RoboDK station: UR10e.rdk

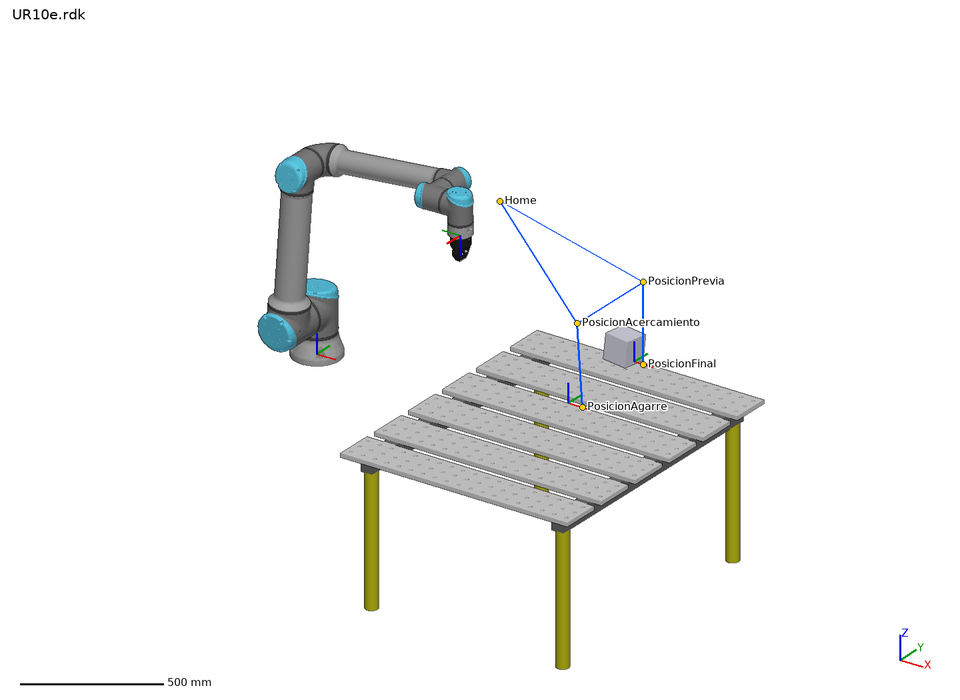
[picture v0: the station drawn from its stored meshes, robots at their saved joint values, targets as dots, program paths as lines]
Station Clase1IndustrialRobotics (saved by RoboDK 5.5.2). Poses are relative to the parent item; angles as X-Y-Z fixed-axis rotations.
  - frame UR10e Base at (0, 0, 0) mm
    - robot UR10e: 6 axes, payload 10 kg, reach 1300 mm, repeatability 0.05 mm, weight 28.9 kg
        modified DH rows (alpha deg, a mm, theta deg, d mm): 0, 0, 0, 180.7; 90, 0, 180, 0; 0, 612.6, 0, 0; 0, 571.335, 0, 174.15; -90, 0, 0, 119.85; 90, 0, 180, 116.55
        joint limits [-360, -360, -360, -360, -360, -360] to [360, 360, 360, 360, 360, 360]; home [0, -90, -90, 0, 90, 0]; saved at [-0.149, -94.095, -80.252, -94.407, 89.966, 1.561]
      - frame RobotiQ 2F85 Base at (0, 0, 0) mm
        - robot RobotiQ 2F85: 1 axes, payload 5 kg
            joint limits [0] to [85]; home [85]; saved at [85]
        - target Open (Cartesian target) at (938.55, 100, 246.18) mm, rotated rx -85.99 ry 0 rz -90 deg; joints [85] of RobotiQ 2F85
        - target Close (Cartesian target) at (0, 0, 103.92) mm; joints [68.98] of RobotiQ 2F85
      - tool 2F85, TCP at (0, 0, 211.5) mm
    - target PosicionAgarre (Cartesian target) at (1059.85, 100, 50) mm, rotated rx -85.99 ry 0 rz -90 deg; joints [21.396, -153.863, -98.022, 76.192, 68.659, -1.57] of UR10e
    - target Home (Cartesian target) at (899.38, -174.15, 913.15) mm, rotated rx -90 ry 0 rz -90 deg; joints [0, -90, -90, 0, 90, 0] of UR10e
    - target PosicionAcercamiento (Cartesian target) at (1037.47, 100, 369.22) mm, rotated rx -85.99 ry 0 rz -90 deg; joints [22.067, -125.528, -106.843, 56.698, 67.99, -1.624] of UR10e
    - target PosicionPrevia (Cartesian target) at (1037.47, 500, 369.22) mm, rotated rx -85.99 ry 0 rz -90 deg; joints [46.712, -135.658, -86.279, 47.776, 43.437, -4.247] of UR10e
    - target PosicionFinal (Cartesian target) at (1037.47, 500, 50) mm, rotated rx -85.99 ry 0 rz -90 deg; joints [46.712, -159.071, -80.316, 65.226, 43.437, -4.247] of UR10e
  - object Table at (1000, 0, 0) mm, rotated rx 0 ry 0 rz 90 deg, size 1193.8 x 965.2 x 609.6 mm, geometry from welding_table.sld
  - frame PosicionA at (1000, 100, 50) mm
  - frame PosicionB at (1000, 500, 50) mm
    - object box at (-40.58, -3.89, 50) mm, rotated rx -4.01 ry 3.72 rz -4.28 deg, size 100 x 100 x 100 mm, geometry from box.sld
  - program ProgramaPrincipal (14 instructions, listed below)
  - Python program CinematicaInversaConGripper (listed below)
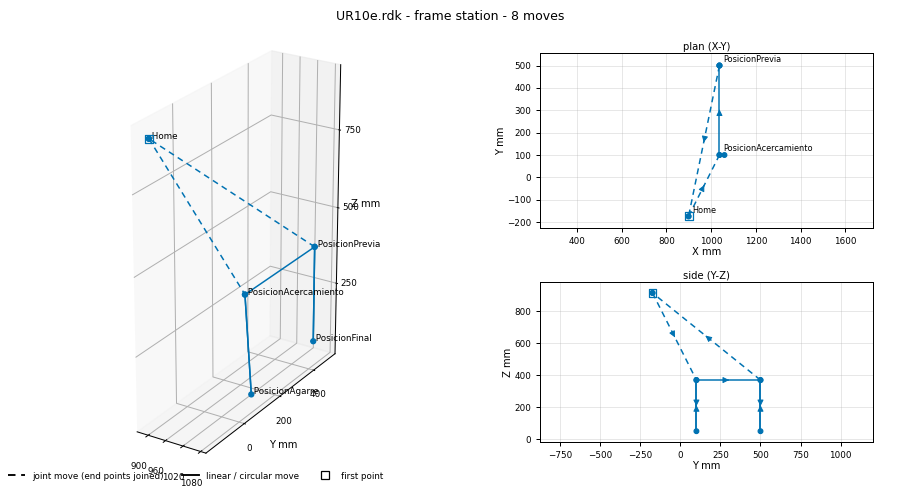
[picture p0: tool path of UR10e.rdk in frame station, 8 of 8 moves have a stored position in this frame; points joined in program order, loops and branches not executed]

--- program ProgramaPrincipal (robot UR10e) ---
  Est. Ref.: UR10e Base
  Est. herr: 2F85
  MoveJ (Home)
  MoveJ (PosicionAcercamiento)
  MoveL (PosicionAgarre)
  Adjuntar a 2F85
  MoveL (PosicionAcercamiento)
  Establecer velocidad (50.0 mm/s)
  MoveL (PosicionPrevia)
  MoveL (PosicionFinal)
  Separar de 2F85
  MoveL (PosicionPrevia)
  Establecer velocidad (500.0 mm/s)
  MoveJ (Home)

--- Python program CinematicaInversaConGripper ---
import math

import numpy as np
from robodk import *
from robolink import *  # RoboDK API
"""
import robotiq_gripper

#from numpy.linalg import inv
#import time

#Funciones para gripper (NO ALTERAR)
def log_info(gripper):
    print(f"Pos: {str(gripper.get_current_position()): >3} "
          f"Open: {gripper.is_open(): <2} "
          f"Closed: {gripper.is_closed(): <2} ")


def dt_gripper_position(current_position): #(NO ALTERAR)
    dt_pos = [0]
    dt_pos[0] = 85 - (current_position / gMax_Pos) * 85
    return dt_pos
"""
# Function to move real gripper and see it in RoboDK simulation (Open) (NO ALTERAR)
def open_gripper():
    if RDK.RunMode() > 1:
        RDK.setRunMode(1) #Set RunMode to see movement in robot and simulation
    time.sleep(0.5)
    gripper.move_and_wait_for_pos(int(gMin_Pos), 255, 255) #Move real gripper
    log_info(gripper) #Print info about gripper position
    dt_pos = dt_gripper_position(gripper.get_current_position()) # give actual position of gripper in milimeters
    dt_gripper.MoveJ(dt_pos) #move simulated gripper
    time.sleep(0.5)
    RDK.setRunMode(6) #Set Run mode to PC-Real Robot connection
    time.sleep(0.5)

# Function to move real gripper and see it in RoboDK simulation (Close) (NO ALTERAR)
def close_gripper():
    if RDK.RunMode() > 1:
        RDK.setRunMode(1)
    gripper.move_and_wait_for_pos(int(gMax_Pos), 255, 191)
    log_info(gripper)
    dt_pos = dt_gripper_position(gripper.get_current_position())
    dt_gripper.MoveJ(dt_pos)
    #input("Press 'Enter' to continue...")
    gripper.move_and_wait_for_pos(gMax_Pos, 255, 191)
    log_info(gripper)
    dt_pos = dt_gripper_position(gripper.get_current_position())
    dt_gripper.MoveJ(dt_pos)
    #input("Press 'Enter' to continue...")
    time.sleep(0.5)
    RDK.setRunMode(6)
    time.sleep(0.5)

#Suministar los datos de posicion y rotacion ROLL PITCH YAW
#TCP: Vector Tool Pose
#X : Posicion en X -- en milimetros [mm]
#Y : Posicion en Y -- en milimetros [mm]
#Z : Posicion en Z -- en milimetros [mm]
#RX : Rotacion en X - Yaw -- En grados [°]
#RY : Rotacion en Y - Pitch -- En grados [°]
#RZ : Rotacion en Z - Roll -- En grados [°]
#VTCP = [X,Y,Z,RX,RY,RZ]

VTCP=[1000,300,500,90,-90,90] #Ejemplo

#Conexion a RoboDK y robot
robot_ip = "192.168.1.10"  # Replace with your robot ip
rdk_ip = 'localhost'  # Or the explicit ip of the computer running RoboDK
### Connect to the RoboDK API ###
RDK = Robolink(robodk_ip=rdk_ip, port=20500)

rdk_robot = RDK.Item('UR10e')  # retrieve the robot by name
dt_gripper = RDK.Item('RobotiQ 2F85')  # the robotiq gripper inside RoboDK, It is not TCP attached to robot

"""
#Este codigo es ESENCIAL para asegurar la conexion al robot
status, status_msg = rdk_robot.ConnectedState()
while status != ROBOTCOM_READY:
    print(status_msg)
    rdk_robot.Disconnect()
    time.sleep(2)
    try:
        success = rdk_robot.Connect(robot_ip=robot_ip) ##IP UR10e PolyScope
        #success = Robot.Connect(robot_ip="192.168.1.10") ##IP UR10e real
        status, status_msg = rdk_robot.ConnectedState()
    except e:
        print(status_msg)
    if status == ROBOTCOM_READY:
        break

# Uses robotiq_gripper class to connect to gripper via sockets
print("Creating gripper...")
gripper = robotiq_gripper.RobotiqGripper()
print("Connecting to gripper...")
gripper.connect(robot_ip, 63352)  # The port on the URe family is 63352
print("Activating gripper...")
# When this executes the gripper will close and open again. Be careful.
# This function gets the max and min values of the gripper
gripper.activate()
# The gripper not always closes using the default max. It depends on the calibration
# So its is useful to know the current max of the system
gMax_Pos = gripper.get_max_position() #Fully Close
gMin_Pos = gripper.get_min_position() #Fully Open
"""
#Longitudes de links
d1= 180.7 #En milimetros
a2 = -612.7 #En mm
a3= -571.55 #En mm
d4= 174.15 #En mm
d5= 119.85 #En mm
d6= 116.55+211.5 #En mm. Se suma el valor del TCP de la herramienta

#Inserte algoritmo de cinematica inversa
def sen(grados):
    return math.sin(math.radians(grados))

def cos(grados):
    return math.cos(math.radians(grados))

def CInversa(VTCP):
    PX=VTCP[0]
    PY=VTCP[1]
    PZ=VTCP[2]
    Psi=VTCP[3]
    Theta=VTCP[4]
    phi=VTCP[5]
    T=np.array([[cos(phi)*cos(Theta),(sen(Psi)*cos(phi)*sen(Theta))-(cos(Psi)*sen(phi)),(sen(Psi)*sen(phi))+(cos(Psi)*cos(phi)*sen(Theta)),PX],
                [cos(Theta)*sen(phi), (cos(Psi)*cos(phi))+(sen(Psi)*sen(phi)*sen(Theta)),(cos(Psi)*sen(phi)*sen(Theta))-(sen(Psi)*cos(phi)),PY],
                [-sen(Theta),sen(Psi)*cos(Theta),cos(Psi)*cos(Theta),PZ],
                [0, 0, 0, 1]])
    for i in range(4):
        for j in range(4):
            T[i][j]=round(T[i][j],2)

    #Calculo del angulo theta1
    #Vector posicion de 0 a 5
    Z06=[T[0][2],T[1][2],T[2][2]]
    P06=[T[0][3],T[1][3],T[2][3]]
    P05=P06-np.dot(d6,Z06) #Se resta a la posicion en el SC6 la distancia al SC5 considerando la rotacion Z06
    phi1=math.degrees(math.atan2(P05[1],P05[0]))
    P05XY=math.sqrt(math.pow(P05[1],2)+math.pow(P05[0],2))
    phi2=math.degrees(math.acos(d4/P05XY))
    theta1=phi1+phi2+90
    theta1=round(theta1,2)
    #INICIO DE CODIGO DE CINEMATICA INVERSA (Del Angulo 2 al 6)
    theta5=math.degrees(math.acos((P06[0]*sen(theta1)-P06[1]*cos(theta1)-d4)/d6))
    CT6=math.degrees(-T[1][0]*sen(theta1)+(T[1][1]*cos(theta1))/sen(theta5))
    ST6=math.degrees(T[0][0]*sen(theta1)-(T[0][1]*cos(theta1))/sen(theta5))
    theta6=math.degrees(math.atan2(CT6,ST6))
    T1=np.array([[cos(theta1),0,sen(theta1),0],[sen(theta1),0,-cos(theta1),0],[0,1,0,d1],[0,0,0,1]])
    T5=np.array([[cos(theta5),0,-sen(theta5),0],[sen(theta5),0,cos(theta5),0],[0,-1,0,d5],[0,0,0,1]])
    T6=np.array([[cos(theta6),-sen(theta6),0,0],[sen(theta6),cos(theta6),0,0],[0,0,1,d6],[0,0,0,1]])
    P45=T5
    P56=T6
    P46=np.dot(P45,P56)
    P64=np.linalg.inv(P46)
    P10=np.linalg.inv(T1)
    P16=np.dot(P10,T)
    P14=np.dot(P16,P64)
    P14XY=math.sqrt((math.pow(P14[1][3],2))+math.pow(P14[0][3],2))
    theta3=math.degrees(math.acos(((P14XY**2)-(a2**2)-(a3**2))/(2*a2*a3)))
    theta2=(math.degrees(math.atan2(-P14[1][3],-P14[0][3])))-math.degrees(math.asin(-a3*sen(theta3)/P14XY))
    T2=np.array([[cos(theta2),-sen(theta2),0,a2*cos(theta2)],[sen(theta2),cos(theta2),0,a2*sen(theta2)],[0,0,1,0],[0,0,0,1]])
    T3=np.array([[cos(theta3),-sen(theta3),0,a3*cos(theta3)],[sen(theta3),cos(theta3),0,a3*sen(theta3)],[0,0,1,0],[0,0,0,1]])
    P12=T2 #CAMBIO
    P23=T3 #CAMBIO
    P13=np.dot(P12,P23)
    P31=np.linalg.inv(P13)
    P34=np.dot(P31,P14)
    theta4=math.degrees(math.atan2(P34[1][0],P34[0][0]))

    #IMPRESION DE CADA ANGULO (NO TOCAR)
    print("\ntheta1:",round(theta1,2))
    print("theta2:",round(theta2,2))
    print("theta3:",round(theta3,2))
    print("theta4:",round(theta4,2))
    print("theta5:",round(theta5,2))
    print("theta6:",round(theta6,2))

    return theta1,theta2,theta3,theta4,theta5,theta6
CInversa(VTCP)
"""
#MOVER AL ROBOT AL PUNTO CALCULADO PARA CORROBORAR
rdk_robot.MoveJ(list(CInversa(VTCP)))
#close_gripper()
#open_gripper()

rdk_robot.Stop()
rdk_robot.Disconnect()
"""
